Staubli VAL3: interfaceDefault.pjx

--- interfaceDefault.pjx ---
Parameters version=s7.11 stackSize=5000 millimeterUnit=true
Program file=ack.pgx
Program file=clearScreen.pgx
Program file=debug.pgx
Program file=feedbackStatus.pgx
Program file=init.pgx
Program file=motionBuffer.pgx
Program file=motionProgress.pgx
Program file=motionStatus.pgx
Program file=start.pgx
Program file=stop.pgx
Program file=trajBuffer.pgx
Program file=velOverwrite.pgx
Data file=interfaceDefault.dtx
Library alias=libQueueFuncs path=Disk://ros_libs/QueueFuncs/QueueFuncs.pjx

--- start.pgx ---
program start()
begin

  // Blank interface library to load at runtime
  // The correct library will be loaded in the application

end

--- ack.pgx ---
public program ack(num x_nHeaderTime, num x_nElapsedTime)
begin

  // Do nothing
  // See start() program for more details

end

--- clearScreen.pgx ---
public program clearScreen()
begin

  // Do nothing
  // See start() program for more details

end

--- debug.pgx ---
public program debug(num& x_nExecStatus)
begin

  // Do nothing
  // See start() program for more details

end

--- feedbackStatus.pgx ---
public program feedbackStatus(num x_nOutConnFlag)
begin

  // Do nothing
  // See start() program for more details

end

--- init.pgx ---
public program init()
begin

  // Do nothing
  // See start() program for more details

end

--- motionBuffer.pgx ---
public program motionBuffer(num x_nMovePts, num x_nElems)
begin

  // Do nothing
  // See start() program for more details

end

--- motionProgress.pgx ---
public program motionProgress(num x_nMoveId, num x_nMotProg)
begin

  // Do nothing
  // See start() program for more details

end

--- motionStatus.pgx ---
public program motionStatus(num x_nInConnFlag)
begin

  // Do nothing
  // See start() program for more details

end

--- trajBuffer.pgx ---
public program trajBuffer(num x_nElems, num x_nPtsPopped)
begin

  // Do nothing
  // See start() program for more details

end

--- velOverwrite.pgx ---
public program velOverwrite(bool x_bOverwriteVel)
begin

  // Do nothing
  // See start() program for more details

end
